PROGRAM PRG_CASE_InitialiseDataManual
VAR
	fbCase_InitialiseData		: FB_CASE_InitialiseData;
	
	(* Init function/method declarations*)
	rTrigDataInit		: R_TRIG;
	bDataInit			: BOOL;
	iOuter				: INT;
	iPack				: INT;
	sPackNum			: STRING;
	sOuterNum			: STRING;
	sPackCode			: STRING;
	
	// old variables
	nOuterIndex				: INT;
	nPackIndex				: INT;
	
	(* Inputs *)	
	bExecute 				: BOOL;	(* set TRUE to move Outers *)
	stCTDateTime			: ST_SYSTEM_DateTime;
	stRejectReasonsForCase	: ST_RejectReasonsForCase;
	
	
	(* In/Out *)
	stProductInstruction	: ST_PCM_Status := (sFieldName := 'PCM_Status_name', nOutersPerCase := 50);
	stCACData 				: ST_CAC_Data;	(* Case Queue *)
	
	(* Outputs *)
	bDone					: BOOL;
	bBusy					: BOOL;
	bDoorReject				: BOOL;
	sRejectCode				: T_MaxString;		
	nMasterListCounter		: INT;	
	bCheckDuplicates		: BOOL;
	
END_VAR

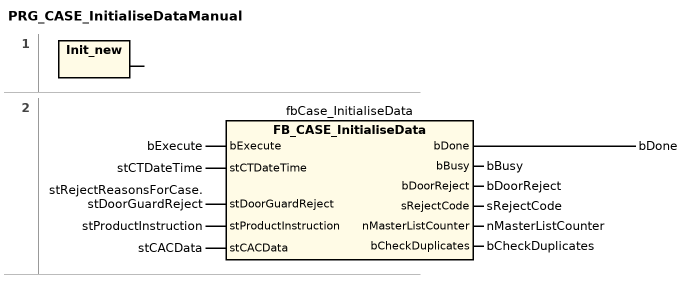
// NETWORK 1
Init_new();

// NETWORK 2
fbCase_InitialiseData(
    bExecute := bExecute,
    stCTDateTime := stCTDateTime,
    stDoorGuardReject := stRejectReasonsForCase.stDoorGuardReject,
    stProductInstruction := stProductInstruction,
    stCACData := stCACData,
    bBusy => bBusy,
    bDoorReject => bDoorReject,
    sRejectCode => sRejectCode,
    nMasterListCounter => nMasterListCounter,
    bCheckDuplicates => bCheckDuplicates); // FB_CASE_InitialiseData
bDone := fbCase_InitialiseData.bDone;

ACTION Init:

rTrigDataInit(CLK := bDataInit);

IF rTrigDataInit.Q THEN
	
	MEMSET(ADR(stCACData), 16#00, SIZEOF(stCACData));	
	
	stProductInstruction.nOutersPerCase 	:= 50;
	stProductInstruction.nPacksPerOuter		:= 10;
	stProductInstruction.nOpMode			:= 11;
	stProductInstruction.sRetailSKU			:= '1234567';
	stProductInstruction.nAcceptanceLevel 	:= 10;


	stCACData.NumberOfOuters			:= stProductInstruction.nOutersPerCase;
	stCACData.CodingAndTrackingMode		:= stProductInstruction.nOpMode;
	stCACData.RetailSKU					:= stProductInstruction.sRetailSKU;

	FOR nOuterIndex := 1 TO stProductInstruction.nOutersPerCase BY 1 DO
	
	stCACData.Outer[nOuterIndex].Barcode 					:= CONCAT('OUTER_', INT_TO_STRING(nOuterIndex));
	stCACData.Outer[nOuterIndex].NumberOfPacks 				:= stProductInstruction.nPacksPerOuter;
	stCACData.Outer[nOuterIndex].NumberOfLinkedPacks 		:= stProductInstruction.nPacksPerOuter;
	stCACData.Outer[nOuterIndex].AcceptanceLevel 			:= stProductInstruction.nAcceptanceLevel;
	stCACData.Outer[nOuterIndex].CodingAndTrackingMode		:= stProductInstruction.nOpMode;
	stCACData.Outer[nOuterIndex].OuterRejectCode			:= 'OK';
	
		FOR  nPackIndex :=1 TO stProductInstruction.nPacksPerOuter BY 1 DO
			stCACData.Outer[nOuterIndex].PackCode[nPackIndex] 		:= F_CONCAT3(stCACData.Outer[nOuterIndex].Barcode,'_PACK_', INT_TO_STRING(nPackIndex));
			IF nPackIndex = 1 THEN
				stCACData.Outer[nOuterIndex].AggregationCodes[1]	:= stCACData.Outer[nOuterIndex].PackCode[nPackIndex];
			END_IF
			IF nPackIndex = 2 THEN
				stCACData.Outer[nOuterIndex].AggregationCodes[2]	:= stCACData.Outer[nOuterIndex].PackCode[nPackIndex];
			END_IF
			stCACData.Outer[nOuterIndex].PackCodeStatus[nPackIndex].5 	:= TRUE;
			stCACData.Outer[nOuterIndex].PackRejectCode[nPackIndex]		:= 'OK';
		END_FOR
	END_FOR	
	
	stCACData.Outer[3].OuterCodeStatus.5 	:= TRUE;
	stCACData.Outer[4].OuterCodeStatus.5	:= TRUE;
	
END_IF
END_ACTION

ACTION Init_new:

rTrigDataInit(CLK := bDataInit);

IF rTrigDataInit.Q THEN
	
	MEMSET(ADR(stCACData), 16#00, SIZEOF(stCACData));	
	
	stProductInstruction.nOutersPerCase 	:= 50;
	stProductInstruction.nPacksPerOuter		:= 10;
	stProductInstruction.nOpMode			:= 11;
	stProductInstruction.sRetailSKU			:= '1234567';
	stProductInstruction.nAcceptanceLevel 	:= 10;


	stCACData.NumberOfOuters			:= stProductInstruction.nOutersPerCase;
	stCACData.CodingAndTrackingMode		:= stProductInstruction.nOpMode;
	stCACData.RetailSKU					:= stProductInstruction.sRetailSKU;

	FOR iOuter := 1 TO stProductInstruction.nOutersPerCase DO
		(* Outer number z zerami *)
		sOuterNum := F_StringAddPrefix(INT_TO_STRING(iOuter),2,'0');
	
		stCACData.Outer[iOuter].Barcode    				:= CONCAT('OUTER', sOuterNum);
		stCACData.Outer[iOuter].NumberOfPacks 			:= stProductInstruction.nPacksPerOuter;
		stCACData.Outer[iOuter].NumberOfLinkedPacks 	:= stProductInstruction.nPacksPerOuter;
		stCACData.Outer[iOuter].AcceptanceLevel 		:= stProductInstruction.nAcceptanceLevel;
		stCACData.Outer[iOuter].CodingAndTrackingMode	:= stProductInstruction.nOpMode;
		stCACData.Outer[iOuter].OuterRejectCode			:= 'OK';
	
		FOR iPack := 1 TO stProductInstruction.nPacksPerOuter DO
			(* Pack number dwucyfrowy z zerami *)
			sPackNum := F_StringAddPrefix(INT_TO_STRING(iPack),2,'0');			
			(* Sklej pack code *)
			sPackCode := CONCAT(CONCAT('PACK', sPackNum), CONCAT('OUTER', sOuterNum));
			
			(* Write Pack Barcodes / Data*)
			stCACData.Outer[iOuter].PackCode[iPack]				:= sPackCode;
			stCACData.Outer[iOuter].PackCodeStatus[iPack]		:= 5;
			stCACData.Outer[iOuter].PackRejectID[iPack]			:= 0;			
			stCACData.Outer[iOuter].PackRejectCode[iPack]		:= 'OK';			
			stCACData.Outer[iOuter].PackCodeStatus[iPack].5 	:= TRUE;
			
			
			IF iPack = 1 THEN
				stCACData.Outer[iOuter].AggregationCodes[1]	:= stCACData.Outer[iOuter].PackCode[iPack];
			END_IF
			IF iPack = 2 THEN
				stCACData.Outer[iOuter].AggregationCodes[2]	:= stCACData.Outer[iOuter].PackCode[iPack];
			END_IF
		END_FOR
	END_FOR	
	
	stCACData.Outer[3].OuterCodeStatus.5 	:= TRUE;
	stCACData.Outer[4].OuterCodeStatus.5	:= TRUE;
	
END_IF
END_ACTION

END_PROGRAM

(* stored: Version 1.1.0.1
   POU PRG_CASE_InitialiseDataManual: Id {9d983551-81c2-4987-8957-1c8f757bfb69}, SpecialFunc None
   Action Init: Id {cfa3d2a8-acd0-4495-8661-28cac742514f}
   Action Init_new: Id {bb6cbe2d-2a6c-4382-84c2-14eb265d8296} *)
